SUBAPPLICATION Ventilsteuerung_Uebung_001_atom (* DigitalInput_I1 auf DigitalOutput_Q1 *)
  (* Standard: 61499-2 *)
  (* Version 1.0, 2023-10-23, franz *)
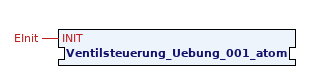
  EVENT_INPUT
    INIT : EInit;
  END_EVENT
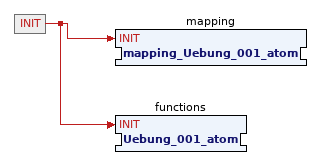
  SUBAPPS
    mapping : mapping_Uebung_001_atom;
    functions : Uebung_001_atom;
  END_SUBAPPS
  EVENT_CONNECTIONS
    INIT TO functions.INIT;
    INIT TO mapping.INIT;
  END_CONNECTIONS
END_SUBAPPLICATION
